// TIA Portal V18 export
TYPE "Cyl"
// stored: IsFailsafeCompliant false
   STRUCT
      In : Struct
         Error : Bool;   // Outer error force output off
         GoWorkInterlock : Bool;   // 1=permit motion
         GoHomeInterlock : Bool;   // 1=permit motion
         WorkPositionSensor : Bool;   // PLC DI
         HomePositionSensor : Bool;   // PLC DI
         ValveType : Bool := true;   // 0 : needn`t holding(2way&3way middle sealing) / 1: need holding(3way middle leaking)
         ManualOutputType : Bool;   // 0 : Output not hold / 1: Output hold (in Manual mode)
         FaultTime : Int := 50;   // Value*100mS
         OnPositionTime : Int := 10;   // Value*100mS
      END_STRUCT;
      Inout : Struct
         ManualGoWork : Bool;
         ManualGoHome : Bool;
         AutoGoWork : Bool;
         AutoGoHome : Bool;
         ResetOut : Bool;   // 泄气
      END_STRUCT;
      S : Struct
         GoWorkTime : Int;
         GoHomeTime : Int;
         WorkFaultTime : Int;
         HomeFaultTime : Int;
         BothSensorOnTime : Int;
         Pulse100mSP : Bool;
         AutoGoWorkP : Bool;
         AutoGoHomeP : Bool;
         GoWork100mSP : Bool;
         GoHome100mSP : Bool;
         BothSensorOn100mSP : Bool;
         Alarm { ExternalVisible := 'False'} : Bool;   // 报警汇总
         spare1 { ExternalVisible := 'False'} : Bool;
         spare2 { ExternalVisible := 'False'} : Byte;
      END_STRUCT;
      Out : Struct
         GoWorkPosition : Bool;   // PLC DQ
         GoHomePosition : Bool;   // PLC DQ
         GoWPButtonActive : Bool;   // For HMI button,indicate can operate go work button
         GoHPButtonActive : Bool;   // For HMI button,indicate can operate go home button
         GoWorkFault : Bool;
         GoHomeFault : Bool;
         SensorPositionFault : Bool;
         CyNO : Byte;
      END_STRUCT;
   END_STRUCT;
END_TYPE
